{attribute addProperty BoxType "AMP8000-0000-0103-0103"}
{attribute addProperty Id "Position_actual_value_invalidAT %I*BOOL812_1st_Additional_position_actual_value_invalidAT %I*BOOL813Ch_A_StatuswordAT %I*UINT1620Ch_A_Position_actual_valueAT %I*DINT3240"}
{attribute addProperty CRC "431710509"}
{attribute addProperty SizeInBites "64"}
{attribute addProperty SizeInBytes "8"}
TYPE Ch_A_AxisMain_Inputs_19BB612D :
STRUCT
	{attribute addProperty Name "Position_actual_value_invalid"}
	Position_actual_value_invalid AT %I* : BOOL;
	{attribute addProperty Name "_1st_Additional_position_actual_value_invalid"}
	_1st_Additional_position_actual_value_invalid AT %I* : BOOL;
	{attribute addProperty Name "Ch_A_Statusword"}
	Ch_A_Statusword AT %I* : UINT;
	{attribute addProperty Name "Ch_A_Position_actual_value"}
	Ch_A_Position_actual_value AT %I* : DINT;
END_STRUCT
END_TYPE

(* stored: Version 1.2.0.0, ProductVersion 3.1.4024.9
   DUT Ch_A_AxisMain_Inputs_19BB612D: Id {8b7b3d78-cb60-4d7c-b45d-76820366eacb} *)
